TYPE STM_Status :
STRUCT
	Status : STM_Status_Status;
END_STRUCT
END_TYPE

(* stored: Version 1.1.0.1, ProductVersion 3.1.4024.3
   DUT STM_Status: Id {c9e27149-420c-426f-9841-4a8ddb9669d3} *)
